// TIA Portal V17 export
// export: Created 2024-08-26T21:07:17.5068745Z, ExportSetting WithDefaults, DisplayName Totally Integrated Automation Portal, DisplayVersion V17 Update 7, DisplayName TIA Portal Openness, DisplayVersion V17 Update 7, DisplayName TIA Portal Version Control Interface, DisplayVersion V17, DisplayName SINAMICS Startdrive Advanced, DisplayVersion V17 SP2, DisplayName SINAMICS Startdrive G110M, G120, G120C, G120D, G120P, G115D, DisplayVersion V17 SP2, DisplayName SINAMICS Startdrive G130, G150, S120, S150, SINAMICS MV, S210, DisplayVersion V17 SP2, DisplayName STEP 7 Professional, DisplayVersion V17 Update 7, DisplayName STEP 7 Safety, DisplayVersion V17 Update 6, DisplayName WinCC Advanced / Unified PC, DisplayVersion V17 Update 7
DATA_BLOCK "CODE READING UPPER"   // DB12
VERSION : 0.1
// stored: AutoNumber true, DBAccessibleFromOPCUA true, DBAccessibleFromWebserver true, InstanceOfName CODE READING, InstanceOfType FB
"CODE READING"
   // VAR_INPUT
   //    hwAdd : HW_IO := 364;
   //    scannerBusy : Bool := FALSE;
   //    autoMode : Bool := FALSE;
   //    manualMode : Bool := TRUE;
   //    scannerReadingComplete : Bool := FALSE;
   //    scannerReadingError : Bool := FALSE;
   //    clearData : Bool := FALSE;
   //    scannerDataSize : Int := 0;
   //    requestScannerAuto : Bool := FALSE;
   //    requestScannerManual : Bool := FALSE;
   //    scannerEnabled : Bool := TRUE;
   //    labelIdentyfier : String[5] := '06';
   //    labelPosition : Int := 4;
   //    labelIdentyfier_2 : String[5] := 'Y4';
   //    labelPosition_2 : Int := 1;
   //    label1 : Bool := FALSE;
   //    label2 : Bool := FALSE;
   // END_VAR
   // VAR_OUTPUT
   //    hmiLabel : String[180] := '';
   //    scannerOk : Bool := FALSE;
   //    scannerOk_2 : Bool := FALSE;
   //    clearReadComplete : Bool := FALSE;
   //    requestScannerOutput : Bool := FALSE;
   //    codeRead : Bool := FALSE;
   // END_VAR
   // VAR
   //    scannerReading { ExternalAccessible := 'False'; ExternalVisible := 'False'; ExternalWritable := 'False'} : Array[0..254] of Char;
   //    ScannerReadTimer { S7_SetPoint := 'True'} : TON_TIME;
   // END_VAR
BEGIN
   scannerReading[0] := '$00';
   scannerReading[1] := 'n';
   scannerReading[2] := '$00';
   scannerReading[3] := 'n';
   scannerReading[4] := '$00';
   scannerReading[5] := 'n';
   scannerReading[6] := '$00';
   scannerReading[7] := '$06';
   scannerReading[8] := 'E';
   scannerReading[9..10] := 'R';
   scannerReading[11] := 'O';
   scannerReading[12] := 'R';
   scannerReading[13] := '$R';
   scannerReading[14..135] := '$00';
   scannerReading[136..254] := ' ';
   ScannerReadTimer.PT := T#50MS;
   ScannerReadTimer.IN := FALSE;
END_DATA_BLOCK
